(*******************************************************************************
                          protoc-gen-twincat V0.0.0.0                           
                  https://github.com/TcHaxx/protoc-gen-twincat                  
*******************************************************************************)
{attribute 'no-analysis'}
{attribute 'pack_mode' := '1'}
// Message with st_prefix and attribute_pack_mode options
TYPE ST_Device :
STRUCT
	name : STRING(256);
	id : DWORD;
	error_codes : ARRAY[0..9] OF WORD;
	error_codes_count : UDINT; // Implict generated field for actual number of items in array error_codes
	temperature : DINT;
	data : ARRAY[0..63] OF BYTE;
	data_count : UDINT; // Implict generated field for actual number of items in array data
END_STRUCT
END_TYPE

(* stored: Version 1.1.0.1
   DUT ST_Device: Id 9684d5b0-0488-4aff-95d0-e68f3364d819 *)
